FUNCTION_BLOCK IlckEnabledManager (* Basic Function Block Type *)
  (* Standard: 61499-2 *)
  (* Version 0.0, 8/14/2024, SESA713705, Schneider Electric, Template *)
  PACKAGE SE.Nereda;
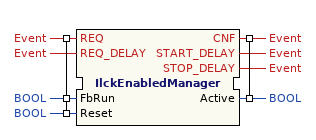
  EVENT_INPUT
    REQ WITH FbRun, Reset;
    REQ_DELAY;
  END_EVENT
  EVENT_OUTPUT
    CNF WITH Active; (* Execution Confirmation *)
    START_DELAY;
    STOP_DELAY;
  END_EVENT
  VAR_INPUT
    FbRun : BOOL;
    Reset : BOOL;
  END_VAR
  VAR_OUTPUT
    Active : BOOL;
  END_VAR
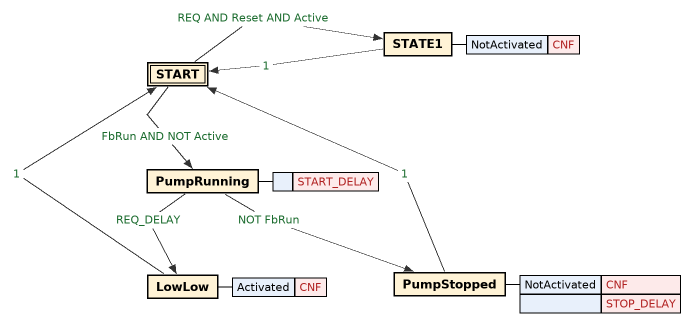
  EC_STATES
    START; (* Initial State *)
    STATE1 : NotActivated -> CNF;
    LowLow : Activated -> CNF;
    PumpRunning : -> START_DELAY;
    PumpStopped : NotActivated -> CNF, -> STOP_DELAY;
  END_STATES
  EC_TRANSITIONS
    START TO PumpRunning := FbRun AND NOT Active;
    START TO STATE1 := REQ AND Reset AND Active;
    LowLow TO START := 1;
    PumpRunning TO LowLow := REQ_DELAY;
    STATE1 TO START := 1;
    PumpRunning TO PumpStopped := NOT FbRun;
    PumpStopped TO START := 1;
  END_TRANSITIONS
  ALGORITHM NotActivated IN ST:
;
Active := FALSE;
  END_ALGORITHM
  ALGORITHM Activated IN ST:
;
Active := TRUE;
  END_ALGORITHM
END_FUNCTION_BLOCK
